// TIA Portal V18 export
DATA_BLOCK "Oscilate_DB"   // DB34
// stored: AutoNumber false, InstanceOfName Oscillate, InstanceOfType FB
"Oscillate"
   // VAR_INPUT
   //    Start : Bool;
   // END_VAR
   // VAR_OUTPUT
   //    FlowmAOut : Real;
   //    TorqmAOut : Real;
   //    EnableP1Fwd : Bool;
   //    EnableP2Fwd : Bool;
   //    EnableP1Rev : Bool;
   //    EnableP2Rev : Bool;
   //    TorqEn : Bool;
   // END_VAR
   // VAR
   //    FlowRev : Bool;
   //    PumpToggle : Bool;
   //    Oscillating : Bool;
   //    Holding : Bool;
   //    OscState : Int;
   //    CalcFlowmA : Real;
   //    LimitFlowmA : Real;
   //    HomePosAbsDeg : Real;
   //    HomePosAbsDegNew : Real;
   //    HomeRelDegNew : Real;
   //    MinmAHigh : Bool;
   //    HoldmALow : Bool;
   //    BumpReactiveTrig : Bool;
   //    BumpFwdTrig : Bool;
   //    BumpRevTrig : Bool;
   //    StartDeg : Real;
   //    HoldFwdFastInc { S7_SetPoint := 'True'} : Bool;
   //    HoldFwdSlowInc : Bool;
   //    HoldFwdFastIDec : Bool;
   //    HoldFwdSlowDev : Bool;
   //    HoldRevFastInc : Bool;
   //    HoldRevSlowInc : Bool;
   //    HoldRevFastIDec : Bool;
   //    HoldRevSlowDev : Bool;
   //    HoldFwdTorqLim : Bool;
   //    HoldRevTorqLim : Bool;
   //    MinSetWarn_TON { S7_SetPoint := 'True'} : TON_TIME;
   //    HoldFWDFast_SlewInc { S7_SetPoint := 'True'} : "SlewInc";
   //    HoldFWDSlow_SlewInc { S7_SetPoint := 'True'} : "SlewInc";
   //    HoldFWDSlow_SlewDec { S7_SetPoint := 'True'} : "SlewDec";
   //    HoldFWDFast_SlewDec { S7_SetPoint := 'True'} : "SlewDec";
   //    HoldFWDTorqLim_TON { S7_SetPoint := 'True'} : TON_TIME;
   //    HoldFwdTorqLim_SlewDec { S7_SetPoint := 'True'} : "SlewDec";
   //    HoldFwdTorqLim_SlewInc { S7_SetPoint := 'True'} : "SlewInc";
   //    HoldRevTorqLim_TON { S7_SetPoint := 'True'} : TON_TIME;
   //    HoldRevTorqLimTrig : Bool;
   //    HoldFwdTorqLimTrig { ExternalAccessible := 'False'; ExternalVisible := 'False'; ExternalWritable := 'False'} : Bool;
   //    HoldRevTorqLim_SlewDec { S7_SetPoint := 'True'} : "SlewDec";
   //    HoldRevTorqLim_SlewInc { S7_SetPoint := 'True'} : "SlewInc";
   //    HoldRevFast_SlewInc { S7_SetPoint := 'True'} : "SlewInc";
   //    HoldRevSlow_SlewInc { S7_SetPoint := 'True'} : "SlewInc";
   //    HoldRevSlow_SlewDec { S7_SetPoint := 'True'} : "SlewDec";
   //    HoldRevFast_SlewDec { S7_SetPoint := 'True'} : "SlewDec";
   //    OscFwdTorqLim { S7_SetPoint := 'True'} : Bool;
   //    OscRevTorqLim : Bool;
   //    OscFwdTrig : Bool;
   //    OscRevTrig : Bool;
   //    HMIBumpFwdLast : Bool;
   //    HMIBumpRevLast : Bool;
   //    HMIBumpReactLast : Bool;
   //    OscFwdAbsDeg : Real;
   //    OscFwdAbsSlowdown : Real;
   //    OscRevAbsDeg : Real;
   //    OscRevAbsSlowdown : Real;
   //    OscFWDTorqLim_TON { S7_SetPoint := 'True'} : TON_TIME;
   //    OscFwdTorqLimTrig : Bool;
   //    OscFwdTorqLim_SlewDec { S7_SetPoint := 'True'} : "SlewDec";
   //    OscFwdTorqLim_SlewInc { S7_SetPoint := 'True'} : "SlewInc";
   //    OscFWDFast_SlewInc { S7_SetPoint := 'True'} : "SlewInc";
   //    OscFWDSlow_SlewInc { S7_SetPoint := 'True'} : "SlewInc";
   //    OscFWDSlow_SlewDec { S7_SetPoint := 'True'} : "SlewDec";
   //    OscFWDFast_SlewDec { S7_SetPoint := 'True'} : "SlewDec";
   //    OscRevTorqLim_TON { S7_SetPoint := 'True'} : TON_TIME;
   //    OscRevTorqLimTrig : Bool;
   //    OscRevTorqLim_SlewDec { S7_SetPoint := 'True'} : "SlewDec";
   //    OscRevTorqLim_SlewInc { S7_SetPoint := 'True'} : "SlewInc";
   //    OscRevFast_SlewInc { S7_SetPoint := 'True'} : "SlewInc";
   //    OscRevSlow_SlewInc { S7_SetPoint := 'True'} : "SlewInc";
   //    OscRevSlow_SlewDec { S7_SetPoint := 'True'} : "SlewDec";
   //    OscRevFast_SlewDec { S7_SetPoint := 'True'} : "SlewDec";
   //    HomeFwdTrig : Bool;
   //    HomeFwdTorqLim : Bool;
   //    HomeFwdTorqLimTrig : Bool;
   //    HomeFwdTorqLim_SlewDec { S7_SetPoint := 'True'} : "SlewDec";
   //    HomeFWDTorqLim_TON { S7_SetPoint := 'True'} : TON_TIME;
   //    HomeFwdTorqLim_SlewInc { S7_SetPoint := 'True'} : "SlewInc";
   //    HomeFWDFast_SlewInc { S7_SetPoint := 'True'} : "SlewInc";
   //    HomeFWDSlow_SlewInc { S7_SetPoint := 'True'} : "SlewInc";
   //    HomeFWDSlow_SlewDec { S7_SetPoint := 'True'} : "SlewDec";
   //    HomeFWDFast_SlewDec { S7_SetPoint := 'True'} : "SlewDec";
   //    HomeRevTrig : Bool;
   //    HomeRevTorqLim_TON { S7_SetPoint := 'True'} : TON_TIME;
   //    HomeRevTorqLim : Bool;
   //    HomeRevTorqLimTrig : Bool;
   //    HomeRevTorqLim_SlewDec { S7_SetPoint := 'True'} : "SlewDec";
   //    HomeRevTorqLim_SlewInc { S7_SetPoint := 'True'} : "SlewInc";
   //    HomeRevFast_SlewInc { S7_SetPoint := 'True'} : "SlewInc";
   //    HomeRevSlow_SlewInc { S7_SetPoint := 'True'} : "SlewInc";
   //    HomeRevSlow_SlewDec { S7_SetPoint := 'True'} : "SlewDec";
   //    HomeRevFast_SlewDec { S7_SetPoint := 'True'} : "SlewDec";
   //    OscHomeLowAbsDeg : Real;
   //    OscHomeLow2AbsDeg : Real;
   //    OscHomeHighAbsDeg : Real;
   //    OscHomeHigh2AbsDeg : Real;
   // END_VAR
BEGIN
END_DATA_BLOCK
